ABB RobotStudio station: LearningSolution_20201010-151018.rsstn

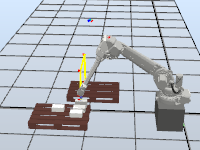
Station LearningSolution (saved by RobotStudio 20.2.9116.0)
Controller LearningController1, task T_ROB1: task frame (RAPID world) sits at (316.67, 323.87, 500) mm in the station
Controller LearningController1
  mechanical unit ROB_1: IRB4600_20_250_C_01, 6 joints, base frame (0, 0, 0) mm
Layout (positions relative to the parent item):
  - IRB4600_20_250_C_01 [mechanism, from Robots\IRB4600_20_250_C_G_01.rslib] at (316.67, 323.87, 500) mm; joint values [-0.1065, 1.0484, 0.0474, 0, 0.475, 3.0351] (rad or m)
  - Base [part] at (57.41, 707.37, 0) mm, rotated rx 90 ry 0 rz 0 deg
  - Euro Pallet from [graphiccomponentgroup, from Equipment\Euro Pallet.rslib] at (1956.13, 0, 0) mm
    - Body 1 [part, from Equipment\Euro Pallet.rslib]
  - Box [part] at (2148.54, 79.91, 246.45) mm
  - Box_2 [part] at (2173.15, 266.46, 244.24) mm, rotated rx -90 ry 0 rz 0 deg
  - Box_3 [part] at (2215.66, 466.33, 244.24) mm, rotated rx -90 ry 0 rz 0 deg
  - Box_4 [part] at (2622.54, 269.44, 244.24) mm, rotated rx -90 ry 0 rz 0 deg
  - Euro Pallet to [graphiccomponentgroup, from Equipment\Euro Pallet.rslib] at (1348.12, -1157.59, 0) mm
    - Body 1 [part, from Equipment\Euro Pallet.rslib]
  - small_suction_gripper [mechanism, from Libraries\small_suction_gripper.rslib] at (2148.53, 128.03, 442.15) mm, rotated rx -180 ry 0 rz 0 deg
  - Positioner_2 [smart component, from Components\Positioner.rslib]
      properties: Object=Box; Position=[2.148529 0.078025 0.244977]; Orientation=[0 0 0]; Reference=Global; ReferenceObject=(none)
  - Attacher [smart component, from Components\Attacher.rslib]
      properties: Parent=small_suction_gripper; Flange=0; Child=Box; Mount=false; Offset=[0 0 0]; Orientation=[0 0 0]
  - Detacher [smart component, from Components\Detacher.rslib]
      properties: Child=Box; KeepPosition=true
  - OD1-B100H50I14-S098974 [part] at (2214.97, 180.09, 357.86) mm, rotated rx 0 ry -90 rz 90 deg
  - Connector [part] at (2138.32, 169.59, 382.67) mm, rotated rx 90 ry 0 rz 0 deg
  - Frame_3 [frame] at (0, 0, 121.44) mm
Attachment: small_suction_gripper is attached to IRB4600_20_250_C_01 / Link6
Attachment: Connector is attached to DEFAULT-34
Attachment: OD1-B100H50I14-S098974 is attached to DEFAULT-34
Collision set CollisionSet_1: Box, Box_2, Box_3, Box_4, Euro Pallet to, Euro Pallet from against , near miss 0 m
Station signals: DI box_positioner
Station logic (signal -> signal, property => property):
  LearningSolution.box_positioner -> Positioner_2.Execute
  LearningController1.att_box -> Attacher.Execute
  LearningController1.det_box -> Detacher.Execute
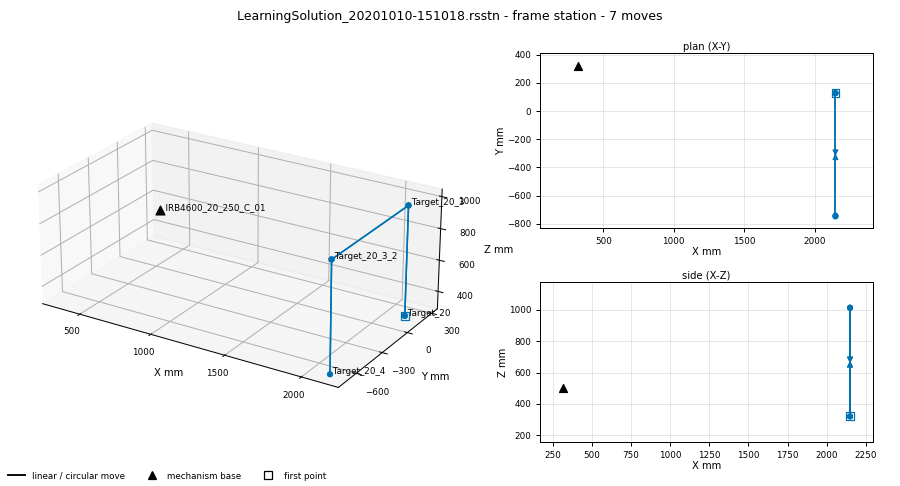
[picture p0: tool path of LearningSolution_20201010-151018.rsstn in frame station, 7 of 7 moves have a stored position in this frame; points joined in program order, loops and branches not executed]
Targets, tools, work objects and paths stored in the station, written as RAPID:
! task T_ROB1
MODULE Module1
  CONST robtarget Target_10:=[[1584.284661998,0,1661.782],[0.5,0,0.866025404,0],[-1,0,-1,0],[9E+09,9E+09,9E+09,9E+09,9E+09,9E+09]];
  CONST robtarget Target_20:=[[1831.863,-195.844947055,-179.285709531],[0,1,0,0],[-1,0,1,0],[9E+09,9E+09,9E+09,9E+09,9E+09,9E+09]];
  CONST robtarget Target_20_3:=[[1831.863,-195.844947055,514.351755884],[0,1,0,0],[-1,0,1,0],[9E+09,9E+09,9E+09,9E+09,9E+09,9E+09]];
  CONST robtarget Target_20_3_2:=[[1831.863,-1071.241124521,514.351755884],[0,1,0,0],[-1,0,1,0],[9E+09,9E+09,9E+09,9E+09,9E+09,9E+09]];
  CONST robtarget Target_20_4:=[[1831.863,-1064.881110195,-179.285709531],[0,1,0,0],[-1,0,1,0],[9E+09,9E+09,9E+09,9E+09,9E+09,9E+09]];
  PROC main()
  ENDPROC
  PROC Path_10_2()
    MoveL Target_20,v100,fine,small_suction_gripper\WObj:=wobj0;
    PulseDO att_box;
    WaitTime 1;
    MoveL Target_20_3,v100,fine,small_suction_gripper\WObj:=wobj0;
    MoveL Target_20_3_2,v600,z5,small_suction_gripper\WObj:=wobj0;
    MoveL Target_20_4,v100,fine,small_suction_gripper\WObj:=wobj0;
    PulseDO det_box;
    WaitTime 1;
    MoveL Target_20_3_2,v100,fine,small_suction_gripper\WObj:=wobj0;
    MoveL Target_20_3,v600,z5,small_suction_gripper\WObj:=wobj0;
    MoveL Target_20,v600,z5,small_suction_gripper\WObj:=wobj0;
  ENDPROC
ENDMODULE

! task T_ROB1
MODULE CalibData
  PERS tooldata small_suction_gripper:=[TRUE,[[0,0,121.436],[1,0,0,0]],[1,[0.443,-9.457,69.909],[1,0,0,0],0,0,0]];
ENDMODULE

